FUNCTION alg_g_a_x: REAL
{ S7_Optimized_Access := 'false' }
    VAR_INPUT
        state: STATE;
    END_VAR

BEGIN
    alg_g_a_x := state.curTime;
END_FUNCTION
